// TIA Portal V19 export
DATA_BLOCK "GlobalDB"   // DB2
{ S7_Optimized_Access := 'TRUE' }
// stored: MemoryReserve 100
   VAR
      TagData : "SiemensDataType";
   END_VAR
BEGIN
END_DATA_BLOCK
